// TIA Portal V20 export
TYPE "type_emRelations_em1_cmStatus"
// stored: Access Published, Namespace Unit1
   STRUCT
      cmBtmDirectionCheckSensor { S7_SetPoint := 'True'} : "LBC_typeDigitalSignalControlNode";
      cmRadiusMeasureBtm { ExternalAccessible := 'False'; ExternalVisible := 'False'; ExternalWritable := 'False'} : "LBC_typeAnalogInputControlNode";
      cmRadiusMeasure { ExternalWritable := 'False'} : "LER_typeRadiusMeasureControlNode";
      cmUnwinderBtmAxisB { ExternalAccessible := 'False'; ExternalVisible := 'False'; ExternalWritable := 'False'; S7_SetPoint := 'True'} : "LBC_typeAxis64PosControlNode";
      cmAirShaftBtmOnOff { ExternalAccessible := 'False'; ExternalVisible := 'False'; ExternalWritable := 'False'; S7_SetPoint := 'True'} : "LBC_typeTwoWayActuatorControlNode";
      cmEpcBtm { ExternalAccessible := 'False'; ExternalVisible := 'False'; ExternalWritable := 'False'} : "LER_typeCON600ControlNode";
   END_STRUCT;
   // cmBtmDirectionCheckSensor.commands.reset := FALSE;
   // cmBtmDirectionCheckSensor.commands.simulation := FALSE;
   // cmBtmDirectionCheckSensor.commands.quality := TRUE;
   // cmRadiusMeasureBtm.commands.simulation := FALSE;
   // cmRadiusMeasureBtm.commands.reset := FALSE;
   // cmRadiusMeasureBtm.commands.quality := TRUE;
   // cmRadiusMeasureBtm.monitoring.valid := FALSE;
   // cmRadiusMeasureBtm.monitoring.busy := FALSE;
   // cmRadiusMeasureBtm.monitoring.error := TRUE;
   // cmRadiusMeasureBtm.monitoring.status := 16#8405;
   // cmRadiusMeasureBtm.monitoring.processValue := 0.0;
   // cmRadiusMeasureBtm.monitoring.limitHigh2 := FALSE;
   // cmRadiusMeasureBtm.monitoring.limitHigh1 := FALSE;
   // cmRadiusMeasureBtm.monitoring.limitLow1 := FALSE;
   // cmRadiusMeasureBtm.monitoring.limitLow2 := FALSE;
   // cmRadiusMeasureBtm.monitoring.maxValueReached := FALSE;
   // cmRadiusMeasureBtm.monitoring.minValueReached := TRUE;
   // cmRadiusMeasure.commands.ZeroSet := FALSE;
   // cmRadiusMeasure.commands.Reset := FALSE;
   // cmRadiusMeasure.monitoring.Radius := 39.0;
   // cmRadiusMeasure.monitoring.Diameter := 78.0;
END_TYPE
